{attribute 'linkalways'} 
{attribute 'no_explicit_call' := 'This FB is a CLASS and must be accessed using methods or properties'}
{attribute 'enable_dynamic_creation'}
FUNCTION_BLOCK _Array0to2OfLREAL EXTENDS ArrayDatatypeBase
VAR CONSTANT
	lBound : DINT := 0;
	uBound : DINT := 2;
END_VAR
VAR
	localData : ARRAY [lBound..uBound] OF LREAL;
	activeData : REFERENCE TO ARRAY [lBound..uBound] OF LREAL REF= localData;
	elements : ARRAY [lBound..uBound] OF _LREAL(0.0);
	baseType : _LREAL(0.0);
END_VAR

PROPERTY PUBLIC Address : PVOID
GET
Address := ADR(activeData);
END_GET
END_PROPERTY

PROPERTY PUBLIC BaseDatatype : I_Datatype
GET
BaseDatatype := baseType;
END_GET
END_PROPERTY

METHOD PUBLIC ClearReference
VAR_INPUT
END_VAR
activeData REF= localData;
SetElementReference();
END_METHOD

METHOD PUBLIC Clone : I_Datatype
VAR
    pClone : POINTER TO _Array0to2OfLREAL;
END_VAR
pClone := __NEW(_Array0to2OfLREAL());
pClone^.Value := Value;
Clone := pClone^;
END_METHOD

METHOD FB_init : BOOL
VAR_INPUT
	bInitRetains : BOOL; // if TRUE, the retain variables are initialized (warm start / cold start)
	bInCopyCode : BOOL;  // if TRUE, the instance afterwards gets moved into the copy code (online change)
END_VAR
SetElementReference();
END_METHOD

METHOD PUBLIC GetElementAsDatatypeByIndex : I_Datatype
VAR_INPUT
	Index : DINT;
END_VAR
GetElementAsDatatypeByIndex := elements[Index];
END_METHOD

METHOD PUBLIC GetElementByIndex : REFERENCE TO _LREAL;
VAR_INPUT
	Index : DINT;
END_VAR
GetElementByIndex REF= elements[Index];
END_METHOD

PROPERTY PUBLIC LowerBound : DINT
GET
LowerBound := lBound;
END_GET
END_PROPERTY

METHOD PUBLIC MakeReferenceTo
VAR_INPUT
	ReferenceTarget : REFERENCE TO ARRAY [lBound..uBound] OF LREAL;
END_VAR
activeData REF= ReferenceTarget;
SetElementReference();
END_METHOD

METHOD PROTECTED OnSerializeArrayValues
VAR_INPUT
	Serializer : I_Serializer;
END_VAR
VAR
	i : DINT;
END_VAR
FOR i := lBound TO uBound DO
	elements[i].SerializeWith(Serializer);
END_FOR
END_METHOD

METHOD PROTECTED SetElementReference
VAR_INPUT
END_VAR
VAR
	i : DINT;
END_VAR
FOR i := lBound TO uBound DO
	elements[i].MakeReferenceTo(activeData[i]);
END_FOR
END_METHOD

PROPERTY PUBLIC Size : UDINT
GET
Size := SIZEOF(activeData);
END_GET
END_PROPERTY

METHOD PROTECTED TryDeserializeArrayValues : BOOL
VAR_INPUT
	Deserializer : I_Deserializer;
	Feedback : I_DeserializerFeedback;
END_VAR
VAR
	enumerator : I_DeserializerArrayForwardEnumerator;
	i : DINT;
END_VAR
enumerator := Deserializer.GetArrayEnumerator();
i := lBound;

WHILE enumerator.MoveNext() AND i <= uBound DO
	
	IF NOT elements[i].TryDeserializeFrom(enumerator.Current, Feedback) THEN
		EXIT;
	END_IF
	i := i + 1;

END_WHILE
enumerator.Dispose();
END_METHOD

METHOD TryMakeReferenceTo : BOOL
VAR_INPUT
	Target : I_Datatype;
END_VAR
VAR
	targetAsArray : I_ArrayDatatype;
	pTargetData : POINTER TO ARRAY [lBound..uBound] OF LREAL;
END_VAR
IF NOT Target.TryResolveAsArrayDatatype(targetAsArray) THEN
	RETURN;
END_IF

IF NOT (targetAsArray.Identifier = Identifier) THEN
	RETURN;
END_IF

pTargetData := Target.Address;
activeData REF= pTargetData^;
SetElementReference();
TryMakeReferenceTo := TRUE;
END_METHOD

PROPERTY PUBLIC UpperBound : DINT
GET
UpperBound := ubound;
END_GET
END_PROPERTY

PROPERTY PUBLIC Value : REFERENCE TO ARRAY [lBound..uBound] OF LREAL;
GET
Value ref= activeData;
END_GET
END_PROPERTY

END_FUNCTION_BLOCK

(* stored: Version 1.1.0.1, ProductVersion 3.1.4024.13
   POU _Array0to2OfLREAL: Id {9d380b32-3610-0bc4-2019-6c5e25a3aa16}, SpecialFunc None
   Folder Core: Id {ff233905-fd73-0c1c-25a3-fb95f39ebfb1}
   Folder Constructor: Id {adf7a95a-ecde-07fe-145e-3c7e59d8be4c}
   Folder Protected: Id {b0272ab4-e9e6-0998-3a97-93912245c8d7}
   Folder Customize: Id {f2870487-a827-004a-287a-ceb27a21e64b}
   Property Address: Id {4d6081c5-2396-0b3c-050d-600f39f7a70a}
   Get Get: Id {b91e1bac-f2c5-03bb-213f-479c9d6e9c9b}
   Property BaseDatatype: Id {56e0ba7b-cefe-0eb9-3afe-2278716ad7b1}
   Get Get: Id {fa4134fc-d3f0-0a6b-1d2c-bc59e367d218}
   Method ClearReference: Id {0bda0615-d482-03f0-3a98-c0fce3174eb6}
   Method Clone: Id {8a98e5e4-6b48-0979-0473-baf08bcf9e97}
   Method FB_init: Id {f4383ff7-bfc8-0e59-0f68-43719aedaee5}
   Method GetElementAsDatatypeByIndex: Id {4922e9f8-c9a1-0d84-08bc-4936c666155f}
   Method GetElementByIndex: Id {4701b97b-7cb7-0519-0138-b99fa94ccf8d}
   Property LowerBound: Id {7ab01210-1fd8-0d75-19ee-f55e0e05c4cb}
   Get Get: Id {270b935d-0a59-09c7-1908-3ad22221995f}
   Method MakeReferenceTo: Id {12c17128-655e-001d-174a-a2b61e4307fc}
   Method OnSerializeArrayValues: Id {cbe0943b-c1ec-004f-3b49-abb8fa4ac023}
   Method SetElementReference: Id {24954636-ca0b-0bb6-3263-8d1e291f8903}
   Property Size: Id {7e4f30df-b60f-0078-3f1d-6f0aea18e48e}
   Get Get: Id {074eb707-305e-0e99-28e9-bc492499d974}
   Method TryDeserializeArrayValues: Id {da752bc1-cd37-036e-3629-9590a0329dfa}
   Method TryMakeReferenceTo: Id {9405b493-b3cf-00bb-3c87-a780d9ce003c}
   Property UpperBound: Id {7d1c51a9-03f3-0286-1bd2-b300452752b4}
   Get Get: Id {ce092675-df12-0c4b-188a-9d0997ab35d1}
   Property Value: Id {fd14ec9b-ce94-0bf9-1948-24fcf47478f2}
   Get Get: Id {c1dccd54-0277-0a0d-1afe-ee7ee37a01c3} *)
